PROGRAM MAIN_Task2
VAR
	MachineSettingsClient : T_MachineSettingsClient; // Receives settings and loaded status from MachineSettingsServer running in separate context (task)
END_VAR

MachineSettingsClient.HandleNotifications();

END_PROGRAM

(* stored: Version 1.1.0.1, ProductVersion 3.1.4024.12
   POU MAIN_Task2: Id {ea8d16ae-7106-48b1-bb65-8de4d17f5cd8}, SpecialFunc None *)
